// TIA Portal V17 export
// export: Created 2025-05-06T14:26:20.7208923Z, ExportSetting WithDefaults, DisplayName Totally Integrated Automation Portal, DisplayVersion V17 Update 8, DisplayName TIA Portal Openness, DisplayVersion V17 Update 8, DisplayName TIA Portal Version Control Interface, DisplayVersion V17, DisplayName SINAMICS Startdrive Advanced, DisplayVersion V17 SP2, DisplayName SINAMICS Startdrive G110M, G120, G120C, G120D, G120P, G115D, DisplayVersion V17 SP2, DisplayName SINAMICS Startdrive G130, G150, S120, S150, SINAMICS MV, S210, DisplayVersion V17 SP2, DisplayName STEP 7 Professional, DisplayVersion V17 Update 8, DisplayName SINUMERIK ONE STEP 7 Toolbox, DisplayVersion V17 Update 12, DisplayName SINUMERIK 840D sl STEP 7 Toolbox, DisplayVersion V17 Update 12, DisplayName STEP 7 Safety, DisplayVersion V17 Update 6, DisplayName WinCC Advanced, DisplayVersion V17 Update 8
FUNCTION "FC7260_HMI_LUBRICATION_GREASE_CONTROL" : Void   // FC7260, LAD
{ S7_Optimized_Access := 'FALSE' }
AUTHOR : ETXETAR
VERSION : 1.0
// stored: AutoNumber false, IsIECCheckEnabled false, SetENOAutomatically false, UDAEnableTagReadback false
   VAR_TEMP
      ERROR_CODE : Int;
      DATA_TIME : Date_And_Time;
      T1 : Bool;
      ERROR_CODE_CONTR_OFF : Int;
      ERROR_CODE_CONTR_ON : Int;
      DATA_TIME_CONTROL_OFF : Date_And_Time;   // DATA TIME WHEN CONTROL OFF
      DATA_TIME_CONTROL_ON : Date_And_Time;   // DATA TIME WHEN CONTROL ON
      DATA_TIME_DIFFERENCE : LTime;   // DATA TIME DIFERENCE
      NUMBER_OF_DAYS : Int;   // NUMBER OF DAYS
   END_VAR
   VAR CONSTANT
      FC_NUMBER : DInt := 7227;
      NUMBER_OF_DAYS_1 : Int := 6;   // NUMBER OF DAYS
   END_VAR
   VAR_TEMP   // added for the SCL form of the ladder/FBD networks
      _w1 : Bool;
   END_VAR
BEGIN

REGION Network 1: READ DATE AND TIME
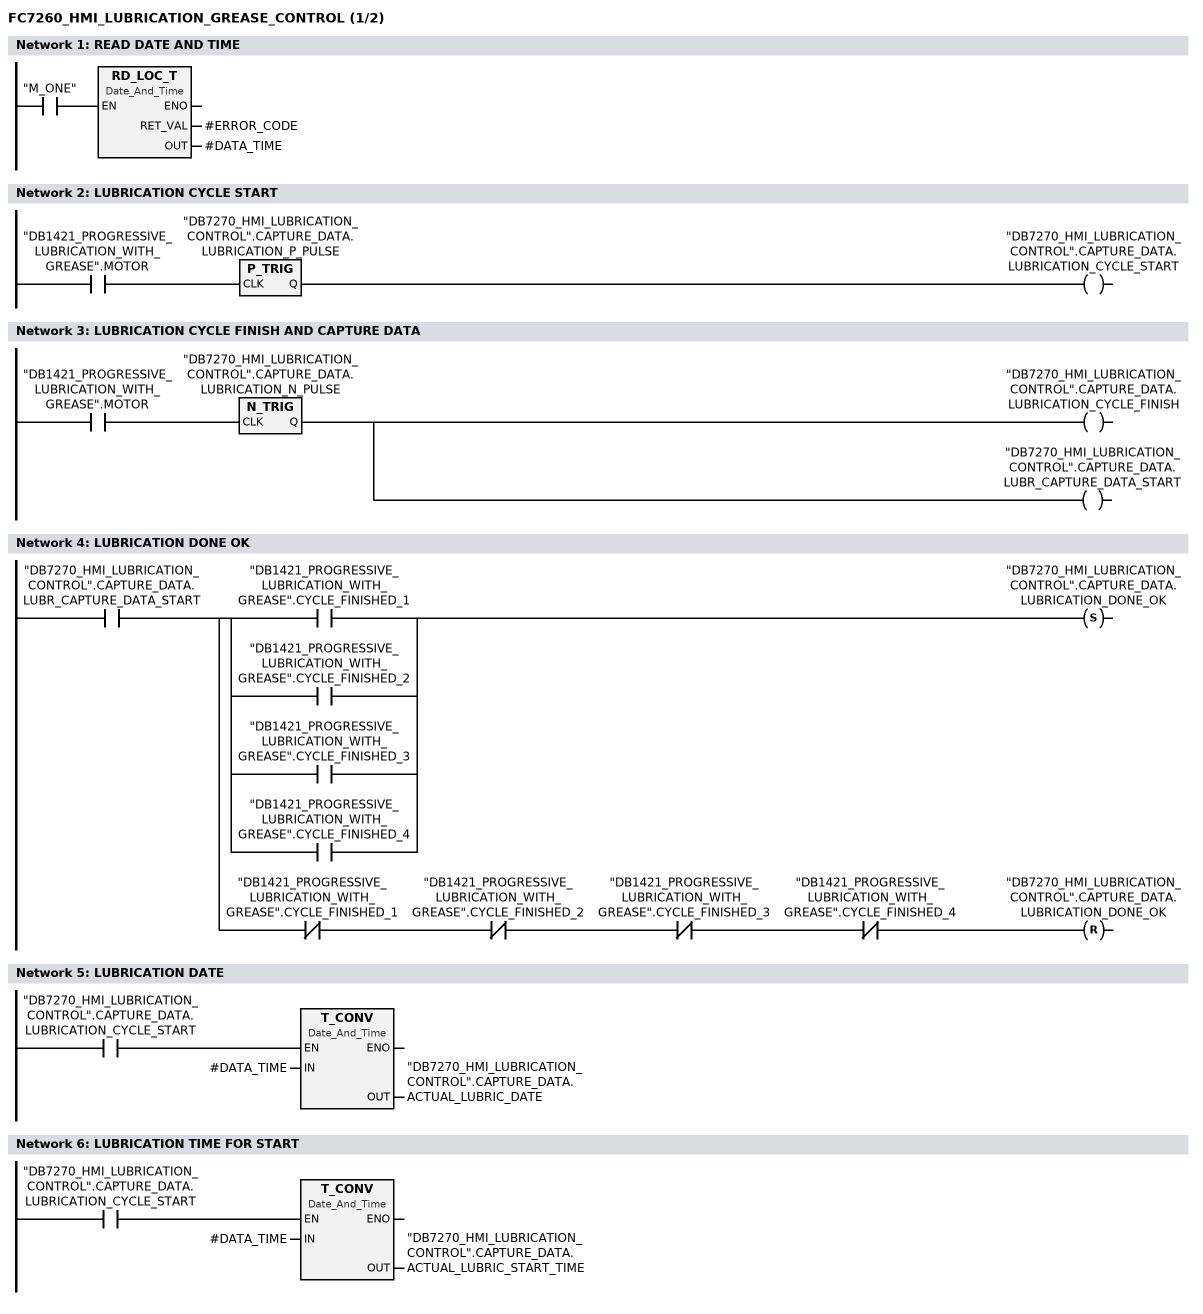
   RUNG wire#powerrail
      Contact( "M_ONE" )
      { S7_Templates := "date_type := Date_And_Time" } RD_LOC_T(RET_VAL => #ERROR_CODE, OUT => #DATA_TIME)
   END_RUNG
   // the same network as SCL:
   IF "M_ONE" THEN #ERROR_CODE := RD_LOC_T(OUT => #DATA_TIME); END_IF;
END_REGION

REGION Network 2: LUBRICATION CYCLE START
   RUNG wire#powerrail
      Contact( "DB1421_PROGRESSIVE_LUBRICATION_WITH_GREASE".MOTOR )
      P_Trig( "DB7270_HMI_LUBRICATION_CONTROL".CAPTURE_DATA.LUBRICATION_P_PULSE )
      Coil( "DB7270_HMI_LUBRICATION_CONTROL".CAPTURE_DATA.LUBRICATION_CYCLE_START )
   END_RUNG
   // the same network as SCL:
   #_w1 := "DB1421_PROGRESSIVE_LUBRICATION_WITH_GREASE".MOTOR AND NOT "DB7270_HMI_LUBRICATION_CONTROL".CAPTURE_DATA.LUBRICATION_P_PULSE;   // rising edge
   "DB7270_HMI_LUBRICATION_CONTROL".CAPTURE_DATA.LUBRICATION_P_PULSE := "DB1421_PROGRESSIVE_LUBRICATION_WITH_GREASE".MOTOR;
   "DB7270_HMI_LUBRICATION_CONTROL".CAPTURE_DATA.LUBRICATION_CYCLE_START := #_w1;
END_REGION

REGION Network 3: LUBRICATION CYCLE FINISH AND CAPTURE DATA
   RUNG wire#powerrail
      Contact( "DB1421_PROGRESSIVE_LUBRICATION_WITH_GREASE".MOTOR )
      N_Trig( "DB7270_HMI_LUBRICATION_CONTROL".CAPTURE_DATA.LUBRICATION_N_PULSE )
      wire#w1
      Coil( "DB7270_HMI_LUBRICATION_CONTROL".CAPTURE_DATA.LUBRICATION_CYCLE_FINISH )
   END_RUNG
   RUNG wire#w1
      Coil( "DB7270_HMI_LUBRICATION_CONTROL".CAPTURE_DATA.LUBR_CAPTURE_DATA_START )
   END_RUNG
   // the same network as SCL:
   #_w1 := NOT "DB1421_PROGRESSIVE_LUBRICATION_WITH_GREASE".MOTOR AND "DB7270_HMI_LUBRICATION_CONTROL".CAPTURE_DATA.LUBRICATION_N_PULSE;   // falling edge
   "DB7270_HMI_LUBRICATION_CONTROL".CAPTURE_DATA.LUBRICATION_N_PULSE := "DB1421_PROGRESSIVE_LUBRICATION_WITH_GREASE".MOTOR;
   "DB7270_HMI_LUBRICATION_CONTROL".CAPTURE_DATA.LUBRICATION_CYCLE_FINISH := #_w1;
   "DB7270_HMI_LUBRICATION_CONTROL".CAPTURE_DATA.LUBR_CAPTURE_DATA_START := #_w1;
END_REGION

REGION Network 4: LUBRICATION DONE OK
   RUNG wire#powerrail
      Contact( "DB7270_HMI_LUBRICATION_CONTROL".CAPTURE_DATA.LUBR_CAPTURE_DATA_START )
      wire#w1
      Contact( "DB1421_PROGRESSIVE_LUBRICATION_WITH_GREASE".CYCLE_FINISHED_1 )
      wire#w2
      S_Coil( "DB7270_HMI_LUBRICATION_CONTROL".CAPTURE_DATA.LUBRICATION_DONE_OK )
   END_RUNG
   RUNG wire#w1
      Contact( "DB1421_PROGRESSIVE_LUBRICATION_WITH_GREASE".CYCLE_FINISHED_2 )
   END_RUNG wire#w2
   RUNG wire#w1
      Contact( "DB1421_PROGRESSIVE_LUBRICATION_WITH_GREASE".CYCLE_FINISHED_3 )
   END_RUNG wire#w2
   RUNG wire#w1
      Contact( "DB1421_PROGRESSIVE_LUBRICATION_WITH_GREASE".CYCLE_FINISHED_4 )
   END_RUNG wire#w2
   RUNG wire#w1
      I_Contact( "DB1421_PROGRESSIVE_LUBRICATION_WITH_GREASE".CYCLE_FINISHED_1 )
      I_Contact( "DB1421_PROGRESSIVE_LUBRICATION_WITH_GREASE".CYCLE_FINISHED_2 )
      I_Contact( "DB1421_PROGRESSIVE_LUBRICATION_WITH_GREASE".CYCLE_FINISHED_3 )
      I_Contact( "DB1421_PROGRESSIVE_LUBRICATION_WITH_GREASE".CYCLE_FINISHED_4 )
      R_Coil( "DB7270_HMI_LUBRICATION_CONTROL".CAPTURE_DATA.LUBRICATION_DONE_OK )
   END_RUNG
   // the same network as SCL:
   IF "DB7270_HMI_LUBRICATION_CONTROL".CAPTURE_DATA.LUBR_CAPTURE_DATA_START AND ("DB1421_PROGRESSIVE_LUBRICATION_WITH_GREASE".CYCLE_FINISHED_1 OR "DB1421_PROGRESSIVE_LUBRICATION_WITH_GREASE".CYCLE_FINISHED_2 OR "DB1421_PROGRESSIVE_LUBRICATION_WITH_GREASE".CYCLE_FINISHED_3 OR "DB1421_PROGRESSIVE_LUBRICATION_WITH_GREASE".CYCLE_FINISHED_4) THEN
       "DB7270_HMI_LUBRICATION_CONTROL".CAPTURE_DATA.LUBRICATION_DONE_OK := TRUE;
   END_IF;
   IF "DB7270_HMI_LUBRICATION_CONTROL".CAPTURE_DATA.LUBR_CAPTURE_DATA_START AND NOT "DB1421_PROGRESSIVE_LUBRICATION_WITH_GREASE".CYCLE_FINISHED_1 AND NOT "DB1421_PROGRESSIVE_LUBRICATION_WITH_GREASE".CYCLE_FINISHED_2 AND NOT "DB1421_PROGRESSIVE_LUBRICATION_WITH_GREASE".CYCLE_FINISHED_3 AND NOT "DB1421_PROGRESSIVE_LUBRICATION_WITH_GREASE".CYCLE_FINISHED_4 THEN
       "DB7270_HMI_LUBRICATION_CONTROL".CAPTURE_DATA.LUBRICATION_DONE_OK := FALSE;
   END_IF;
END_REGION

REGION Network 5: LUBRICATION DATE
   RUNG wire#powerrail
      Contact( "DB7270_HMI_LUBRICATION_CONTROL".CAPTURE_DATA.LUBRICATION_CYCLE_START )
      { S7_Templates := "[src_type := Date_And_Time, dest_type := Date]" } T_CONV(IN := #DATA_TIME, OUT => "DB7270_HMI_LUBRICATION_CONTROL".CAPTURE_DATA.ACTUAL_LUBRIC_DATE)
   END_RUNG
   // the same network as SCL:
   IF "DB7270_HMI_LUBRICATION_CONTROL".CAPTURE_DATA.LUBRICATION_CYCLE_START THEN
       T_CONV(IN := #DATA_TIME, OUT => "DB7270_HMI_LUBRICATION_CONTROL".CAPTURE_DATA.ACTUAL_LUBRIC_DATE);
   END_IF;
END_REGION

REGION Network 6: LUBRICATION TIME FOR START
   RUNG wire#powerrail
      Contact( "DB7270_HMI_LUBRICATION_CONTROL".CAPTURE_DATA.LUBRICATION_CYCLE_START )
      { S7_Templates := "[src_type := Date_And_Time, dest_type := Time_Of_Day]" } T_CONV(IN := #DATA_TIME, OUT => "DB7270_HMI_LUBRICATION_CONTROL".CAPTURE_DATA.ACTUAL_LUBRIC_START_TIME)
   END_RUNG
   // the same network as SCL:
   IF "DB7270_HMI_LUBRICATION_CONTROL".CAPTURE_DATA.LUBRICATION_CYCLE_START THEN
       T_CONV(IN := #DATA_TIME, OUT => "DB7270_HMI_LUBRICATION_CONTROL".CAPTURE_DATA.ACTUAL_LUBRIC_START_TIME);
   END_IF;
END_REGION

REGION Network 7: LUBRICATION TIME FOR FINISH
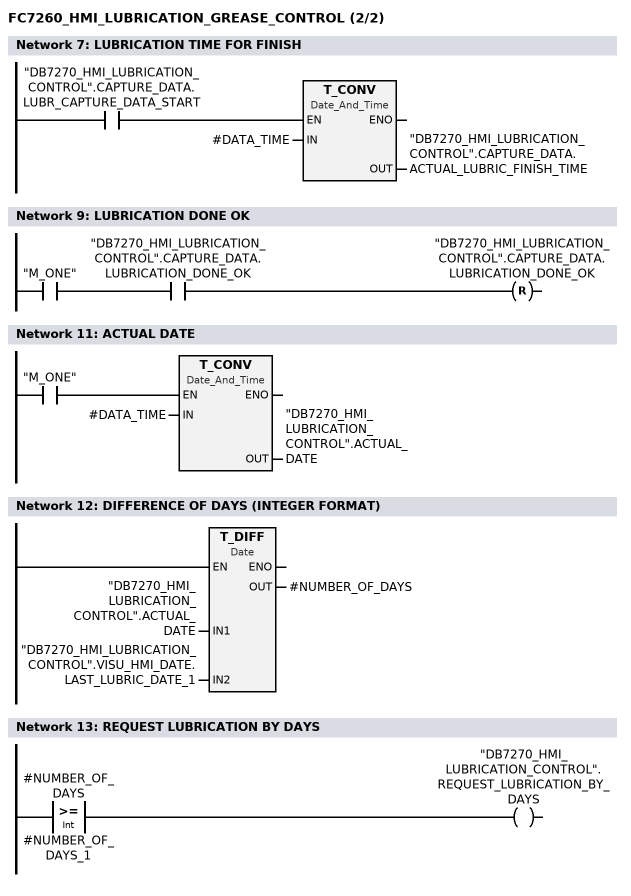
   RUNG wire#powerrail
      Contact( "DB7270_HMI_LUBRICATION_CONTROL".CAPTURE_DATA.LUBR_CAPTURE_DATA_START )
      { S7_Templates := "[src_type := Date_And_Time, dest_type := Time_Of_Day]" } T_CONV(IN := #DATA_TIME, OUT => "DB7270_HMI_LUBRICATION_CONTROL".CAPTURE_DATA.ACTUAL_LUBRIC_FINISH_TIME)
   END_RUNG
   // the same network as SCL:
   IF "DB7270_HMI_LUBRICATION_CONTROL".CAPTURE_DATA.LUBR_CAPTURE_DATA_START THEN
       T_CONV(IN := #DATA_TIME, OUT => "DB7270_HMI_LUBRICATION_CONTROL".CAPTURE_DATA.ACTUAL_LUBRIC_FINISH_TIME);
   END_IF;
END_REGION

NETWORK
TITLE = READ TIME
      A     "DB7270_HMI_LUBRICATION_CONTROL".CAPTURE_DATA.LUBR_CAPTURE_DATA_START;
      JCN   END;

// DATE
      L     "DB7270_HMI_LUBRICATION_CONTROL".VISU_HMI_DATE.LAST_LUBRIC_DATE_9;
      T     "DB7270_HMI_LUBRICATION_CONTROL".VISU_HMI_DATE.LAST_LUBRIC_DATE_10;
      L     "DB7270_HMI_LUBRICATION_CONTROL".VISU_HMI_DATE.LAST_LUBRIC_DATE_8;
      T     "DB7270_HMI_LUBRICATION_CONTROL".VISU_HMI_DATE.LAST_LUBRIC_DATE_9;
      L     "DB7270_HMI_LUBRICATION_CONTROL".VISU_HMI_DATE.LAST_LUBRIC_DATE_7;
      T     "DB7270_HMI_LUBRICATION_CONTROL".VISU_HMI_DATE.LAST_LUBRIC_DATE_8;
      L     "DB7270_HMI_LUBRICATION_CONTROL".VISU_HMI_DATE.LAST_LUBRIC_DATE_6;
      T     "DB7270_HMI_LUBRICATION_CONTROL".VISU_HMI_DATE.LAST_LUBRIC_DATE_7;
      L     "DB7270_HMI_LUBRICATION_CONTROL".VISU_HMI_DATE.LAST_LUBRIC_DATE_5;
      T     "DB7270_HMI_LUBRICATION_CONTROL".VISU_HMI_DATE.LAST_LUBRIC_DATE_6;
      L     "DB7270_HMI_LUBRICATION_CONTROL".VISU_HMI_DATE.LAST_LUBRIC_DATE_4;
      T     "DB7270_HMI_LUBRICATION_CONTROL".VISU_HMI_DATE.LAST_LUBRIC_DATE_5;
      L     "DB7270_HMI_LUBRICATION_CONTROL".VISU_HMI_DATE.LAST_LUBRIC_DATE_3;
      T     "DB7270_HMI_LUBRICATION_CONTROL".VISU_HMI_DATE.LAST_LUBRIC_DATE_4;
      L     "DB7270_HMI_LUBRICATION_CONTROL".VISU_HMI_DATE.LAST_LUBRIC_DATE_2;
      T     "DB7270_HMI_LUBRICATION_CONTROL".VISU_HMI_DATE.LAST_LUBRIC_DATE_3;
      L     "DB7270_HMI_LUBRICATION_CONTROL".VISU_HMI_DATE.LAST_LUBRIC_DATE_1;
      T     "DB7270_HMI_LUBRICATION_CONTROL".VISU_HMI_DATE.LAST_LUBRIC_DATE_2;
      L     "DB7270_HMI_LUBRICATION_CONTROL".CAPTURE_DATA.ACTUAL_LUBRIC_DATE;
      T     "DB7270_HMI_LUBRICATION_CONTROL".VISU_HMI_DATE.LAST_LUBRIC_DATE_1;

// START TIME

      L     "DB7270_HMI_LUBRICATION_CONTROL".VISU_HMI_TIME_START.LAST_LUBRIC_START_TIME_9;
      T     "DB7270_HMI_LUBRICATION_CONTROL".VISU_HMI_TIME_START.LAST_LUBRIC_START_TIME_10;
      L     "DB7270_HMI_LUBRICATION_CONTROL".VISU_HMI_TIME_START.LAST_LUBRIC_START_TIME_8;
      T     "DB7270_HMI_LUBRICATION_CONTROL".VISU_HMI_TIME_START.LAST_LUBRIC_START_TIME_9;
      L     "DB7270_HMI_LUBRICATION_CONTROL".VISU_HMI_TIME_START.LAST_LUBRIC_START_TIME_7;
      T     "DB7270_HMI_LUBRICATION_CONTROL".VISU_HMI_TIME_START.LAST_LUBRIC_START_TIME_8;
      L     "DB7270_HMI_LUBRICATION_CONTROL".VISU_HMI_TIME_START.LAST_LUBRIC_START_TIME_6;
      T     "DB7270_HMI_LUBRICATION_CONTROL".VISU_HMI_TIME_START.LAST_LUBRIC_START_TIME_7;
      L     "DB7270_HMI_LUBRICATION_CONTROL".VISU_HMI_TIME_START.LAST_LUBRIC_START_TIME_5;
      T     "DB7270_HMI_LUBRICATION_CONTROL".VISU_HMI_TIME_START.LAST_LUBRIC_START_TIME_6;
      L     "DB7270_HMI_LUBRICATION_CONTROL".VISU_HMI_TIME_START.LAST_LUBRIC_START_TIME_4;
      T     "DB7270_HMI_LUBRICATION_CONTROL".VISU_HMI_TIME_START.LAST_LUBRIC_START_TIME_5;
      L     "DB7270_HMI_LUBRICATION_CONTROL".VISU_HMI_TIME_START.LAST_LUBRIC_START_TIME_3;
      T     "DB7270_HMI_LUBRICATION_CONTROL".VISU_HMI_TIME_START.LAST_LUBRIC_START_TIME_4;
      L     "DB7270_HMI_LUBRICATION_CONTROL".VISU_HMI_TIME_START.LAST_LUBRIC_START_TIME_2;
      T     "DB7270_HMI_LUBRICATION_CONTROL".VISU_HMI_TIME_START.LAST_LUBRIC_START_TIME_3;
      L     "DB7270_HMI_LUBRICATION_CONTROL".VISU_HMI_TIME_START.LAST_LUBRIC_START_TIME_1;
      T     "DB7270_HMI_LUBRICATION_CONTROL".VISU_HMI_TIME_START.LAST_LUBRIC_START_TIME_2;
      L     "DB7270_HMI_LUBRICATION_CONTROL".CAPTURE_DATA.ACTUAL_LUBRIC_START_TIME;
      T     "DB7270_HMI_LUBRICATION_CONTROL".VISU_HMI_TIME_START.LAST_LUBRIC_START_TIME_1;

// FINISH TIME

      L     "DB7270_HMI_LUBRICATION_CONTROL".VISU_HMI_TIME_FINISH.LAST_LUBRIC_FINISH_TIME_9;
      T     "DB7270_HMI_LUBRICATION_CONTROL".VISU_HMI_TIME_FINISH.LAST_LUBRIC_FINISH_TIME_10;
      L     "DB7270_HMI_LUBRICATION_CONTROL".VISU_HMI_TIME_FINISH.LAST_LUBRIC_FINISH_TIME_8;
      T     "DB7270_HMI_LUBRICATION_CONTROL".VISU_HMI_TIME_FINISH.LAST_LUBRIC_FINISH_TIME_9;
      L     "DB7270_HMI_LUBRICATION_CONTROL".VISU_HMI_TIME_FINISH.LAST_LUBRIC_FINISH_TIME_7;
      T     "DB7270_HMI_LUBRICATION_CONTROL".VISU_HMI_TIME_FINISH.LAST_LUBRIC_FINISH_TIME_8;
      L     "DB7270_HMI_LUBRICATION_CONTROL".VISU_HMI_TIME_FINISH.LAST_LUBRIC_FINISH_TIME_6;
      T     "DB7270_HMI_LUBRICATION_CONTROL".VISU_HMI_TIME_FINISH.LAST_LUBRIC_FINISH_TIME_7;
      L     "DB7270_HMI_LUBRICATION_CONTROL".VISU_HMI_TIME_FINISH.LAST_LUBRIC_FINISH_TIME_5;
      T     "DB7270_HMI_LUBRICATION_CONTROL".VISU_HMI_TIME_FINISH.LAST_LUBRIC_FINISH_TIME_6;
      L     "DB7270_HMI_LUBRICATION_CONTROL".VISU_HMI_TIME_FINISH.LAST_LUBRIC_FINISH_TIME_4;
      T     "DB7270_HMI_LUBRICATION_CONTROL".VISU_HMI_TIME_FINISH.LAST_LUBRIC_FINISH_TIME_5;
      L     "DB7270_HMI_LUBRICATION_CONTROL".VISU_HMI_TIME_FINISH.LAST_LUBRIC_FINISH_TIME_3;
      T     "DB7270_HMI_LUBRICATION_CONTROL".VISU_HMI_TIME_FINISH.LAST_LUBRIC_FINISH_TIME_4;
      L     "DB7270_HMI_LUBRICATION_CONTROL".VISU_HMI_TIME_FINISH.LAST_LUBRIC_FINISH_TIME_2;
      T     "DB7270_HMI_LUBRICATION_CONTROL".VISU_HMI_TIME_FINISH.LAST_LUBRIC_FINISH_TIME_3;
      L     "DB7270_HMI_LUBRICATION_CONTROL".VISU_HMI_TIME_FINISH.LAST_LUBRIC_FINISH_TIME_1;
      T     "DB7270_HMI_LUBRICATION_CONTROL".VISU_HMI_TIME_FINISH.LAST_LUBRIC_FINISH_TIME_2;
      L     "DB7270_HMI_LUBRICATION_CONTROL".CAPTURE_DATA.ACTUAL_LUBRIC_FINISH_TIME;
      T     "DB7270_HMI_LUBRICATION_CONTROL".VISU_HMI_TIME_FINISH.LAST_LUBRIC_FINISH_TIME_1;

//DONE

      A     "DB7270_HMI_LUBRICATION_CONTROL".VISU_HMI_DONE.LUBRI_STATUS_DONE_9;
      =     "DB7270_HMI_LUBRICATION_CONTROL".VISU_HMI_DONE.LUBRI_STATUS_DONE_10;
      A     "DB7270_HMI_LUBRICATION_CONTROL".VISU_HMI_DONE.LUBRI_STATUS_DONE_8;
      =     "DB7270_HMI_LUBRICATION_CONTROL".VISU_HMI_DONE.LUBRI_STATUS_DONE_9;
      A     "DB7270_HMI_LUBRICATION_CONTROL".VISU_HMI_DONE.LUBRI_STATUS_DONE_7;
      =     "DB7270_HMI_LUBRICATION_CONTROL".VISU_HMI_DONE.LUBRI_STATUS_DONE_8;
      A     "DB7270_HMI_LUBRICATION_CONTROL".VISU_HMI_DONE.LUBRI_STATUS_DONE_6;
      =     "DB7270_HMI_LUBRICATION_CONTROL".VISU_HMI_DONE.LUBRI_STATUS_DONE_7;
      A     "DB7270_HMI_LUBRICATION_CONTROL".VISU_HMI_DONE.LUBRI_STATUS_DONE_5;
      =     "DB7270_HMI_LUBRICATION_CONTROL".VISU_HMI_DONE.LUBRI_STATUS_DONE_6;
      A     "DB7270_HMI_LUBRICATION_CONTROL".VISU_HMI_DONE.LUBRI_STATUS_DONE_4;
      =     "DB7270_HMI_LUBRICATION_CONTROL".VISU_HMI_DONE.LUBRI_STATUS_DONE_5;
      A     "DB7270_HMI_LUBRICATION_CONTROL".VISU_HMI_DONE.LUBRI_STATUS_DONE_3;
      =     "DB7270_HMI_LUBRICATION_CONTROL".VISU_HMI_DONE.LUBRI_STATUS_DONE_4;
      A     "DB7270_HMI_LUBRICATION_CONTROL".VISU_HMI_DONE.LUBRI_STATUS_DONE_2;
      =     "DB7270_HMI_LUBRICATION_CONTROL".VISU_HMI_DONE.LUBRI_STATUS_DONE_3;
      A     "DB7270_HMI_LUBRICATION_CONTROL".VISU_HMI_DONE.LUBRI_STATUS_DONE_1;
      =     "DB7270_HMI_LUBRICATION_CONTROL".VISU_HMI_DONE.LUBRI_STATUS_DONE_2;
      A     "DB7270_HMI_LUBRICATION_CONTROL".CAPTURE_DATA.LUBRICATION_DONE_OK;
      =     "DB7270_HMI_LUBRICATION_CONTROL".VISU_HMI_DONE.LUBRI_STATUS_DONE_1;
END:  NOP   0;


REGION Network 9: LUBRICATION DONE OK
   RUNG wire#powerrail
      Contact( "M_ONE" )
      Contact( "DB7270_HMI_LUBRICATION_CONTROL".CAPTURE_DATA.LUBRICATION_DONE_OK )
      R_Coil( "DB7270_HMI_LUBRICATION_CONTROL".CAPTURE_DATA.LUBRICATION_DONE_OK )
   END_RUNG
   // the same network as SCL:
   IF "M_ONE" AND "DB7270_HMI_LUBRICATION_CONTROL".CAPTURE_DATA.LUBRICATION_DONE_OK THEN
       "DB7270_HMI_LUBRICATION_CONTROL".CAPTURE_DATA.LUBRICATION_DONE_OK := FALSE;
   END_IF;
END_REGION

REGION Network 10: ************** NUMBER OF DAYS BETWEEN THE LAST LUBRICATION **************
   // If no lubrication has been done in one week (6 days)
END_REGION

REGION Network 11: ACTUAL DATE
   RUNG wire#powerrail
      Contact( "M_ONE" )
      { S7_Templates := "[src_type := Date_And_Time, dest_type := Date]" } T_CONV(IN := #DATA_TIME, OUT => "DB7270_HMI_LUBRICATION_CONTROL".ACTUAL_DATE)
   END_RUNG
   // the same network as SCL:
   IF "M_ONE" THEN T_CONV(IN := #DATA_TIME, OUT => "DB7270_HMI_LUBRICATION_CONTROL".ACTUAL_DATE); END_IF;
END_REGION

REGION Network 12: DIFFERENCE OF DAYS (INTEGER FORMAT)
   RUNG wire#powerrail
      { S7_Templates := "[date_type := Date, time_type := Int]" } T_DIFF(IN1 := "DB7270_HMI_LUBRICATION_CONTROL".ACTUAL_DATE, IN2 := "DB7270_HMI_LUBRICATION_CONTROL".VISU_HMI_DATE.LAST_LUBRIC_DATE_1, OUT => #NUMBER_OF_DAYS)
   END_RUNG
   // the same network as SCL:
   T_DIFF(IN1 := "DB7270_HMI_LUBRICATION_CONTROL".ACTUAL_DATE,
          IN2 := "DB7270_HMI_LUBRICATION_CONTROL".VISU_HMI_DATE.LAST_LUBRIC_DATE_1,
          OUT => #NUMBER_OF_DAYS);
END_REGION

REGION Network 13: REQUEST LUBRICATION BY DAYS
   RUNG wire#powerrail
      { S7_Templates := "SrcType := Int" } GE_Contact(in1 := #NUMBER_OF_DAYS, in2 := #NUMBER_OF_DAYS_1)
      Coil( "DB7270_HMI_LUBRICATION_CONTROL".REQUEST_LUBRICATION_BY_DAYS )
   END_RUNG
   // the same network as SCL:
   "DB7270_HMI_LUBRICATION_CONTROL".REQUEST_LUBRICATION_BY_DAYS := #NUMBER_OF_DAYS >= #NUMBER_OF_DAYS_1;
END_REGION
END_FUNCTION
